// TIA Portal V20 export
FUNCTION_BLOCK "LER_ServoPress"   // FB220, LAD
// stored: Access Published, MemoryReserve 100, SetENOAutomatically false
   VAR_INPUT
      enable : Bool;
      enableManualCmds : Bool;
      interlockHome : Bool;
      interlockRunSequence : Bool;
      interlockJogForward : Bool;
      interlockJogBackward : Bool;
   END_VAR
   VAR_OUTPUT
      error : Bool;
      status : Word;
   END_VAR
   VAR_IN_OUT
      configuration : "LER_typeServoPressConfiguration";
      moduleInterface : "LER_typeServoPressInterface";
      controlNode : "LER_typeServoPressControlNode";
   END_VAR
   VAR
      statProfinetInput { ExternalAccessible := 'False'; ExternalVisible := 'False'; ExternalWritable := 'False'} : "LER_typeServoPress20ByteIn";
      statProfinetOutput { ExternalAccessible := 'False'; ExternalVisible := 'False'; ExternalWritable := 'False'} : "LER_typeServoPress20ByteOut";
      statMonitoring { ExternalAccessible := 'False'; ExternalVisible := 'False'; ExternalWritable := 'False'} : "LER_typeServoPressMonitoring";
      statConfig { ExternalAccessible := 'False'; ExternalVisible := 'False'; ExternalWritable := 'False'} : "LER_typeServoPressConfiguration";
      statRetValInt { ExternalAccessible := 'False'; ExternalVisible := 'False'; ExternalWritable := 'False'} : Array[1..#count] of Int;
      statRetValWord { ExternalAccessible := 'False'; ExternalVisible := 'False'; ExternalWritable := 'False'} : Array[1..#count] of Word;
      statTonTimer { ExternalAccessible := 'False'; ExternalVisible := 'False'; ExternalWritable := 'False'} : Array[0..99] of TON_TIME;
      statConfigCheck { ExternalAccessible := 'False'; ExternalVisible := 'False'; ExternalWritable := 'False'} : Array[0..19] of Bool;
      statConfigHold { ExternalAccessible := 'False'; ExternalVisible := 'False'; ExternalWritable := 'False'} : Array[0..19] of Bool;
      statServoAlarm { ExternalAccessible := 'False'; ExternalVisible := 'False'; ExternalWritable := 'False'} : Struct
         alarmState_0 : Array[0..7] of Bool;
         alarmState_1 : Array[0..7] of Bool;
         alarmState_2 : Array[0..7] of Bool;
         alarmState_3 : Array[0..7] of Bool;
         alarmState_4 : Array[0..7] of Bool;
         alarmState_5 : Array[0..7] of Bool;
         alarmState_6 : Array[0..7] of Bool;
         alarmState_7 : Array[0..7] of Bool;
      END_STRUCT;
      statStep { ExternalAccessible := 'False'; ExternalVisible := 'False'; ExternalWritable := 'False'} : Int;
      statConfigBusy { ExternalAccessible := 'False'; ExternalVisible := 'False'; ExternalWritable := 'False'} : Bool;
      statAckCheck { ExternalAccessible := 'False'; ExternalVisible := 'False'; ExternalWritable := 'False'} : Bool;
      statStop { ExternalAccessible := 'False'; ExternalVisible := 'False'; ExternalWritable := 'False'} : Bool;
   END_VAR
   VAR_TEMP
      tempRetVal : Array[1..#count] of Int;
      tempIndex : Int;
      tempSequenceEnd : Bool;
   END_VAR
   VAR CONSTANT
      False : Bool := False;
      delayTime : Time := T#3s;
      count : Int := 2;
      statusNoErrorOccurred : Word := 16#0000;   // No error occurred.
      errStatusAlarm : Word := 16#8000;
      errStatusSeq : Word := 16#8001;
      errStatusServo : Word := 16#8002;
      errHwdNotConfigured : Word := 16#8090;   // You have not configured a module for the specified hardware identifier or You have ignored the restriction concerning the length of consistent data, or you have not specified a hardware identifier as an address at parameter LADDR
      errRecordDataType : Word := 16#8092;   // Non-supported data type in the RECORD parameter.
      errNoDpProfinetIoModule : Word := 16#8093;   // No DP module/PROFINET IO device from which you can read consistent data exists for the hardware identifier specified in LADDR . This error code also occurs if the module addressed by means of LADDR does not have inputs.
      errIoAccessPermission : Word := 16#80A0;   // An access error was detected when accessing the I/O.
      errRecordLengthInsufficient : Word := 16#80B1;   // The length of the specified destination area at parameter RECORD is shorter than the configured user data length.
      errDataNotReceived : Word := 16#80C0;   // The data have not been read yet.
   END_VAR
   // // statServoAlarm.alarmState_0[0] : ALARM_SETUP_MISMATCH
   // // statServoAlarm.alarmState_0[1] : ALARM_X_SENSOR_CALIBRATION
   // // statServoAlarm.alarmState_0[2] : ALARM_Y_SENSOR_CALIBRATION
   // // statServoAlarm.alarmState_0[3] : ALARM_SENSOR_TEST
   // // statServoAlarm.alarmState_0[4] : ALARM_SENSOR_TEST_WARNING
   // // statServoAlarm.alarmState_0[5] : ALARM_OVER_PIEZO_RANGE
   // // statServoAlarm.alarmState_0[6] : ALARM_NO_EO_CONFIGURED
   // // statServoAlarm.alarmState_0[7] : ALARM_SETUO_MISMATCH_WARNING
   // // statServoAlarm.alarmState_1[0] : reserved
   // // statServoAlarm.alarmState_1[1] : reserved
   // // statServoAlarm.alarmState_1[2] : ALARM_INACTIVE_MP_SELECTED
   // // statServoAlarm.alarmState_1[3] : ALARM_NOK_IN_SEQUENCE
   // // statServoAlarm.alarmState_1[4] : ALARM_NOK_IN_SEQUENCE_WARNING
   // // statServoAlarm.alarmState_1[5] : ALARM_LOST_CYCLES
   // // statServoAlarm.alarmState_1[6] : ALARM_LOST_CYCLES_WARNING
   // // statServoAlarm.alarmState_1[7] : ALARM_NOK_PERCENTAGE_EXCEEDED
   // // statServoAlarm.alarmState_2[0] : ALARM_ENVELOPE_TREND
   // // statServoAlarm.alarmState_2[1] : ALARM_ENVELOPE_WARNING
   // // statServoAlarm.alarmState_2[2] : ALARM_SELFTEST_STRAIN_GAGE_NOK
   // // statServoAlarm.alarmState_2[3] : ALARM_DIG_IO_SHORT_CIRCUIT
   // // statServoAlarm.alarmState_2[4] : ALARM_SELFTEST_5V_SENSOR_POWER
   // // statServoAlarm.alarmState_2[5] : ALARM_SELFTEST_24V_SENSOR_POWER
   // // statServoAlarm.alarmState_2[6] : ALARM_SAMBA_NO_NETWORK_WARNING
   // // statServoAlarm.alarmState_2[7] : ALARM_SAMBA_MEMORY_FULL
   // // statServoAlarm.alarmState_3[0] : ALARM_SAMBA_MEMORY_FULL_WARNING
   // // statServoAlarm.alarmState_3[1] : ALARM_MEMORY_CARD_FULL_WARNING
   // // statServoAlarm.alarmState_3[2] : ALARM_FIFO_FULL
   // // statServoAlarm.alarmState_3[3] : ALARM_FIFO_FULL_WARNING
   // // statServoAlarm.alarmState_3[4] : ALARM_READING_UV_WITHOUT_DESCRIPTION
   // // statServoAlarm.alarmState_3[5] : ALARM_POWER_COULD_NOT_BE_ENABLED
   // // statServoAlarm.alarmState_3[6] : ALARM_MULTIPLE_PLC_MOVEMENT_COMMANDS
   // // statServoAlarm.alarmState_3[7] : ALARM_SEQ_CALCULATOR_IN_MEASUREMENT
   // // statServoAlarm.alarmState_4[0] : ALARM_SEQ_DYNAMIC_CALC_DIV_BY_ZERO
   // // statServoAlarm.alarmState_4[1] : ALARM_SEQ_DYNAMIC_FORCE_TRIGGER_NOT_
   // // statServoAlarm.alarmState_4[2] : ALARM_SEQ_POSITION_SET_OUTSIDE_THE_RA
   // // statServoAlarm.alarmState_4[3] : ALARM_SERVO_CONTROLLER_CONNECTION
   // // statServoAlarm.alarmState_4[4] : ALARM_SERVO_CONTROLLER_ERROR
   // // statServoAlarm.alarmState_4[5] : ALARM_SERVO_CONTROLLER_WARNING
   // // statServoAlarm.alarmState_4[6] : ALARM_SERVO_MAX_FORCE_TRIGGER
   // // statServoAlarm.alarmState_4[7] : ALARM_SERVO_DISPL_OVERRANGE
   // // statServoAlarm.alarmState_5[0] : ALARM_SERVO_STOP_EXT_SIGNAL_NOT_REACHED
   // // statServoAlarm.alarmState_5[1] : ALARM_SEQ_DYNAMIC_ZERO_MOTION_SPEED
   // // statServoAlarm.alarmState_5[2] : ALARM_ADC_2_DAC_ADC_FACTOR_IS_OUT_OF_RANGE
   // // statServoAlarm.alarmState_5[3] : ALARM_SEQ_SPEED_SET_OUTSIDE_THE_RANG
   // // statServoAlarm.alarmState_5[4] : ALARM_JOG_SPEED_IS_OUT_OF_RANGE
   // // statServoAlarm.alarmState_5[5] : ALARM_BRAKETEST_FAILED
   // // statServoAlarm.alarmState_5[6] : ALARM_SEQ_DYNAMIC_UNKNOWN_ERROR
   // // statServoAlarm.alarmState_5[7] : ALARM_SEQ_DIGITAL_INPUT_TIMOUT_BEFORE_SIGNAL
   VAR_TEMP   // added for the SCL form of the ladder/FBD networks
      _w1 : Bool;
      _w2 : Bool;
      _w3 : Bool;
   END_VAR
BEGIN

REGION Network 1: DP Read
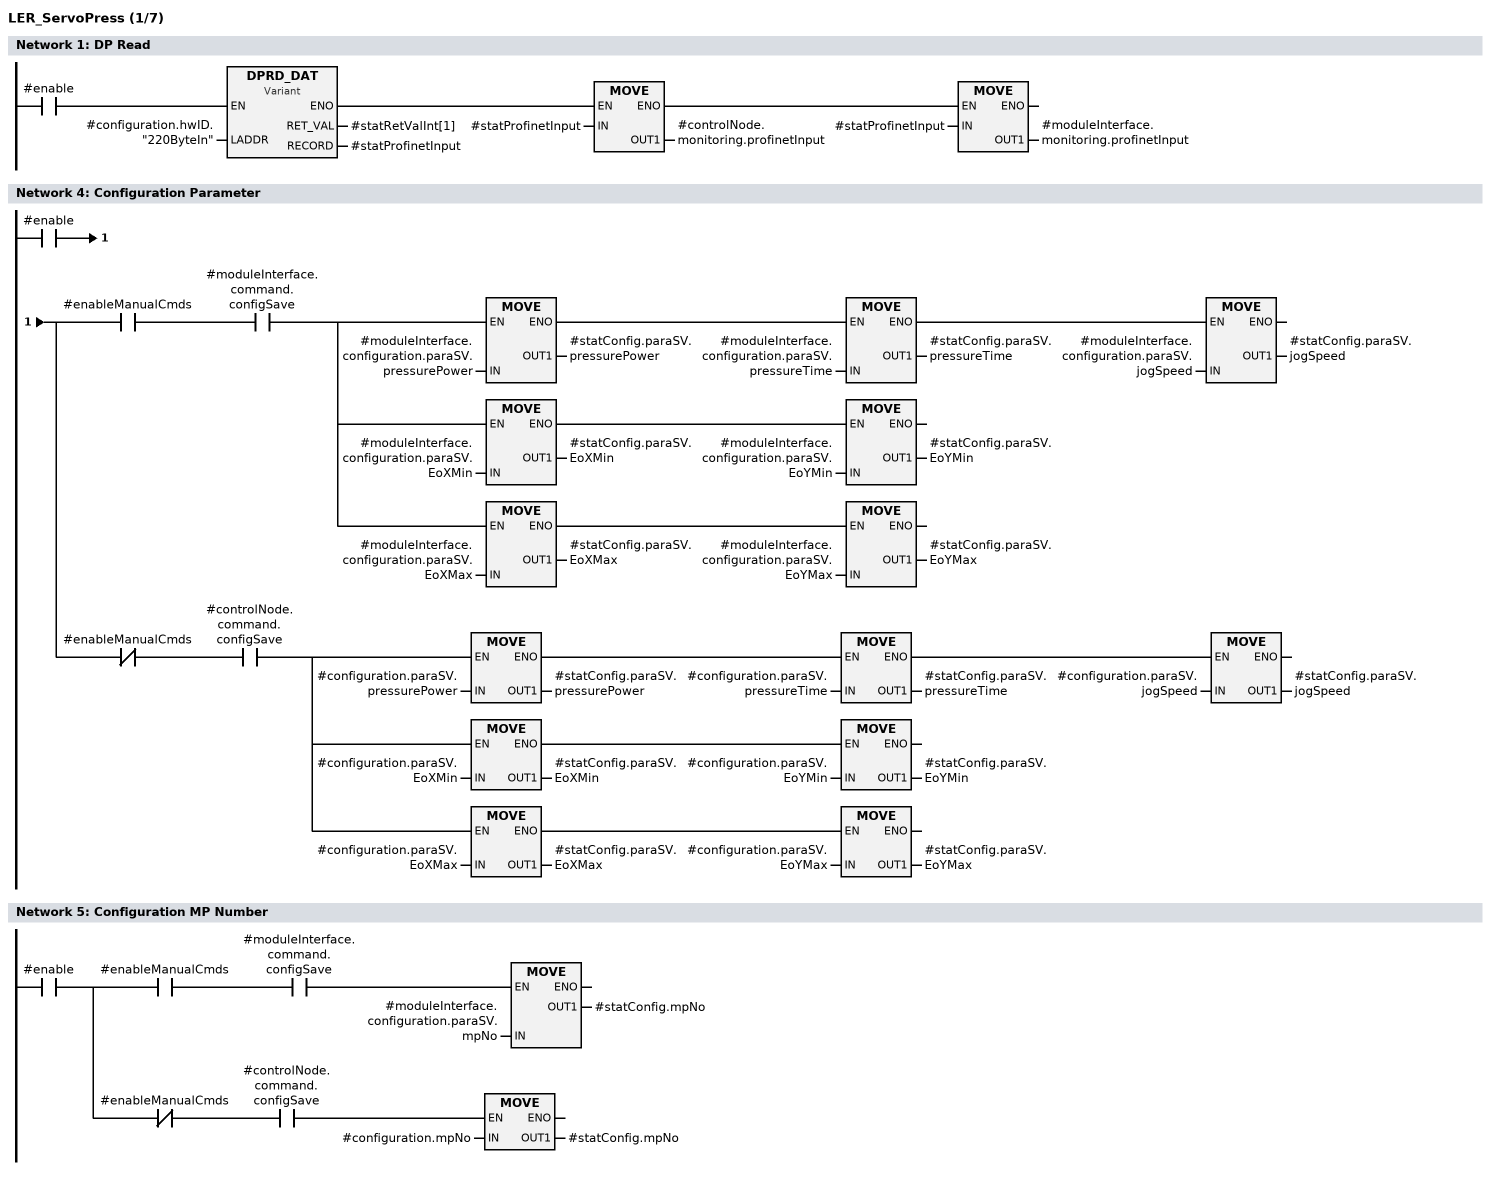
   RUNG wire#powerrail
      Contact( #enable )
      { S7_Templates := "[ptr_type := Variant, laddr_type := HW_IO]" } DPRD_DAT(LADDR := #configuration.hwID."220ByteIn", RET_VAL => #statRetValInt[1], RECORD => #statProfinetInput)
      Move(in := #statProfinetInput, out1 => #controlNode.monitoring.profinetInput)
      Move(in := #statProfinetInput, out1 => #moduleInterface.monitoring.profinetInput)
   END_RUNG
   // the same network as SCL:
   #statRetValInt[1] := DPRD_DAT(EN := #enable,
                           LADDR := #configuration.hwID."220ByteIn",
                           RECORD => #statProfinetInput,
                           ENO => #_w1);
   IF #_w1 THEN
       #controlNode.monitoring.profinetInput := #statProfinetInput;
       #moduleInterface.monitoring.profinetInput := #statProfinetInput;
   END_IF;
END_REGION

REGION Network 2 (SCL): Input Mapping
   REGION Input mapping

   #statMonitoring.profinetInput := #statProfinetInput;

   END_REGION
END_REGION

REGION Network 3 (SCL): Error Status
   REGION Error check

       IF #enable THEN
           IF #statRetValInt <> #tempRetVal THEN
               FOR #tempIndex := 1 TO #count DO
                   #statRetValWord[#tempIndex] := INT_TO_WORD(#statRetValInt[#tempIndex]); // convert the return value of DPRD, DPWR form int to word
                   CASE #statRetValWord[#tempIndex] OF

                       #errHwdNotConfigured:
                           #status := #errHwdNotConfigured;

                       #errRecordDataType:
                           #status := #errRecordDataType;

                       #errNoDpProfinetIoModule:
                           #status := #errNoDpProfinetIoModule;

                       #errIoAccessPermission:
                           #status := #errIoAccessPermission;

                       #errRecordLengthInsufficient:
                           #status := #errRecordLengthInsufficient;

                       #errDataNotReceived:
                           #status := #errDataNotReceived;
                   END_CASE;
               END_FOR;

           ELSIF #statMonitoring.profinetInput.ALARM THEN
               #status := #errStatusAlarm;

           ELSIF #statMonitoring.profinetInput."SEQUENCE-ERROR" THEN
               #status := #errStatusSeq;

           ELSIF #statMonitoring.profinetInput."SERVO-ERROR" THEN
               #status := #errStatusServo;

           ELSE
               #status := #statusNoErrorOccurred;
           END_IF;
       ELSE
           #status := #statusNoErrorOccurred;
       END_IF;

       #error := #status <> 0;

   END_REGION
END_REGION

REGION Network 4: Configuration Parameter
   RUNG wire#powerrail
      Contact( #enable )
      wire#w1
      Contact( #enableManualCmds )
      Contact( #moduleInterface.command.configSave )
      wire#w2
      Move(in := #moduleInterface.configuration.paraSV.pressurePower, out1 => #statConfig.paraSV.pressurePower)
      Move(in := #moduleInterface.configuration.paraSV.pressureTime, out1 => #statConfig.paraSV.pressureTime)
      Move(in := #moduleInterface.configuration.paraSV.jogSpeed, out1 => #statConfig.paraSV.jogSpeed)
   END_RUNG
   RUNG wire#w2
      Move(in := #moduleInterface.configuration.paraSV.EoXMin, out1 => #statConfig.paraSV.EoXMin)
      Move(in := #moduleInterface.configuration.paraSV.EoYMin, out1 => #statConfig.paraSV.EoYMin)
   END_RUNG
   RUNG wire#w2
      Move(in := #moduleInterface.configuration.paraSV.EoXMax, out1 => #statConfig.paraSV.EoXMax)
      Move(in := #moduleInterface.configuration.paraSV.EoYMax, out1 => #statConfig.paraSV.EoYMax)
   END_RUNG
   RUNG wire#w1
      I_Contact( #enableManualCmds )
      Contact( #controlNode.command.configSave )
      wire#w3
      Move(in := #configuration.paraSV.pressurePower, out1 => #statConfig.paraSV.pressurePower)
      Move(in := #configuration.paraSV.pressureTime, out1 => #statConfig.paraSV.pressureTime)
      Move(in := #configuration.paraSV.jogSpeed, out1 => #statConfig.paraSV.jogSpeed)
   END_RUNG
   RUNG wire#w3
      Move(in := #configuration.paraSV.EoXMin, out1 => #statConfig.paraSV.EoXMin)
      Move(in := #configuration.paraSV.EoYMin, out1 => #statConfig.paraSV.EoYMin)
   END_RUNG
   RUNG wire#w3
      Move(in := #configuration.paraSV.EoXMax, out1 => #statConfig.paraSV.EoXMax)
      Move(in := #configuration.paraSV.EoYMax, out1 => #statConfig.paraSV.EoYMax)
   END_RUNG
   // the same network as SCL:
   IF #enable AND #enableManualCmds AND #moduleInterface.command.configSave THEN
       #statConfig.paraSV.pressurePower := #moduleInterface.configuration.paraSV.pressurePower;
       #statConfig.paraSV.pressureTime := #moduleInterface.configuration.paraSV.pressureTime;
       #statConfig.paraSV.jogSpeed := #moduleInterface.configuration.paraSV.jogSpeed;
       #statConfig.paraSV.EoXMin := #moduleInterface.configuration.paraSV.EoXMin;
       #statConfig.paraSV.EoYMin := #moduleInterface.configuration.paraSV.EoYMin;
       #statConfig.paraSV.EoXMax := #moduleInterface.configuration.paraSV.EoXMax;
       #statConfig.paraSV.EoYMax := #moduleInterface.configuration.paraSV.EoYMax;
   END_IF;
   IF #enable AND NOT #enableManualCmds AND #controlNode.command.configSave THEN
       #statConfig.paraSV.pressurePower := #configuration.paraSV.pressurePower;
       #statConfig.paraSV.pressureTime := #configuration.paraSV.pressureTime;
       #statConfig.paraSV.jogSpeed := #configuration.paraSV.jogSpeed;
       #statConfig.paraSV.EoXMin := #configuration.paraSV.EoXMin;
       #statConfig.paraSV.EoYMin := #configuration.paraSV.EoYMin;
       #statConfig.paraSV.EoXMax := #configuration.paraSV.EoXMax;
       #statConfig.paraSV.EoYMax := #configuration.paraSV.EoYMax;
   END_IF;
END_REGION

REGION Network 5: Configuration MP Number
   RUNG wire#powerrail
      Contact( #enable )
      wire#w1
      Contact( #enableManualCmds )
      Contact( #moduleInterface.command.configSave )
      Move(in := #moduleInterface.configuration.paraSV.mpNo, out1 => #statConfig.mpNo)
   END_RUNG
   RUNG wire#w1
      I_Contact( #enableManualCmds )
      Contact( #controlNode.command.configSave )
      Move(in := #configuration.mpNo, out1 => #statConfig.mpNo)
   END_RUNG
   // the same network as SCL:
   IF #enable AND #enableManualCmds AND #moduleInterface.command.configSave THEN
       #statConfig.mpNo := #moduleInterface.configuration.paraSV.mpNo;
   END_IF;
   IF #enable AND NOT #enableManualCmds AND #controlNode.command.configSave THEN
       #statConfig.mpNo := #configuration.mpNo;
   END_IF;
END_REGION

REGION Network 6: Configuration Sequence Number
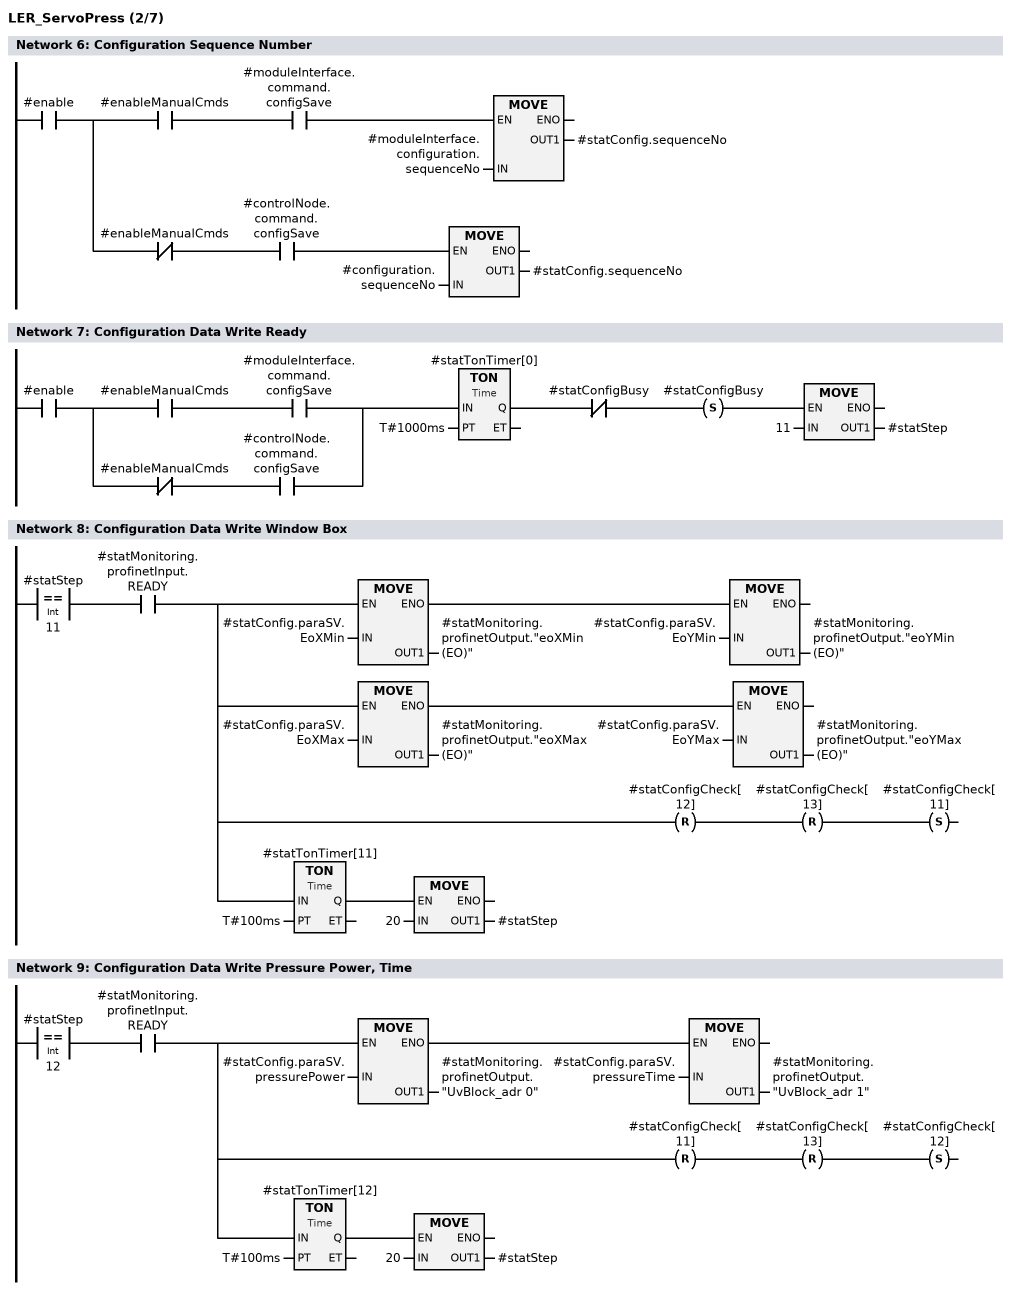
   RUNG wire#powerrail
      Contact( #enable )
      wire#w1
      Contact( #enableManualCmds )
      Contact( #moduleInterface.command.configSave )
      Move(in := #moduleInterface.configuration.sequenceNo, out1 => #statConfig.sequenceNo)
   END_RUNG
   RUNG wire#w1
      I_Contact( #enableManualCmds )
      Contact( #controlNode.command.configSave )
      Move(in := #configuration.sequenceNo, out1 => #statConfig.sequenceNo)
   END_RUNG
   // the same network as SCL:
   IF #enable AND #enableManualCmds AND #moduleInterface.command.configSave THEN
       #statConfig.sequenceNo := #moduleInterface.configuration.sequenceNo;
   END_IF;
   IF #enable AND NOT #enableManualCmds AND #controlNode.command.configSave THEN
       #statConfig.sequenceNo := #configuration.sequenceNo;
   END_IF;
END_REGION

REGION Network 7: Configuration Data Write Ready
   RUNG wire#powerrail
      Contact( #enable )
      wire#w1
      Contact( #enableManualCmds )
      Contact( #moduleInterface.command.configSave )
      wire#w2
      { S7_Templates := "time_type := Time" } #statTonTimer[0].TON(pt := T#1000ms, et =>)
      I_Contact( #statConfigBusy )
      S_Coil( #statConfigBusy )
      Move(in := 11, out1 => #statStep)
   END_RUNG
   RUNG wire#w1
      I_Contact( #enableManualCmds )
      Contact( #controlNode.command.configSave )
   END_RUNG wire#w2
   // the same network as SCL:
   #statTonTimer[0].TON(IN := #enable AND ((#enableManualCmds AND #moduleInterface.command.configSave) OR (NOT #enableManualCmds AND #controlNode.command.configSave)),
                        PT := T#1000ms);
   #_w1 := #statTonTimer[0].Q AND NOT #statConfigBusy;
   IF #_w1 THEN
       #statConfigBusy := TRUE;
       #statStep := 11;
   END_IF;
END_REGION

REGION Network 8: Configuration Data Write Window Box
   RUNG wire#powerrail
      { S7_Templates := "SrcType := Int" } EQ_Contact(in1 := #statStep, in2 := 11)
      Contact( #statMonitoring.profinetInput.READY )
      wire#w1
      Move(in := #statConfig.paraSV.EoXMin, out1 => #statMonitoring.profinetOutput."eoXMin (EO)")
      Move(in := #statConfig.paraSV.EoYMin, out1 => #statMonitoring.profinetOutput."eoYMin (EO)")
   END_RUNG
   RUNG wire#w1
      Move(in := #statConfig.paraSV.EoXMax, out1 => #statMonitoring.profinetOutput."eoXMax (EO)")
      Move(in := #statConfig.paraSV.EoYMax, out1 => #statMonitoring.profinetOutput."eoYMax (EO)")
   END_RUNG
   RUNG wire#w1
      R_Coil( #statConfigCheck[12] )
      R_Coil( #statConfigCheck[13] )
      S_Coil( #statConfigCheck[11] )
   END_RUNG
   RUNG wire#w1
      { S7_Templates := "time_type := Time" } #statTonTimer[11].TON(pt := T#100ms, et =>)
      Move(in := 20, out1 => #statStep)
   END_RUNG
   // the same network as SCL:
   #_w1 := (#statStep = 11) AND #statMonitoring.profinetInput.READY;
   IF #_w1 THEN
       #statMonitoring.profinetOutput."eoXMin (EO)" := #statConfig.paraSV.EoXMin;
       #statMonitoring.profinetOutput."eoYMin (EO)" := #statConfig.paraSV.EoYMin;
       #statMonitoring.profinetOutput."eoXMax (EO)" := #statConfig.paraSV.EoXMax;
       #statMonitoring.profinetOutput."eoYMax (EO)" := #statConfig.paraSV.EoYMax;
       #statConfigCheck[12] := FALSE;
       #statConfigCheck[13] := FALSE;
       #statConfigCheck[11] := TRUE;
   END_IF;
   #statTonTimer[11].TON(IN := #_w1, PT := T#100ms);
   IF #statTonTimer[11].Q THEN #statStep := 20; END_IF;
END_REGION

REGION Network 9: Configuration Data Write Pressure Power, Time
   RUNG wire#powerrail
      { S7_Templates := "SrcType := Int" } EQ_Contact(in1 := #statStep, in2 := 12)
      Contact( #statMonitoring.profinetInput.READY )
      wire#w1
      Move(in := #statConfig.paraSV.pressurePower, out1 => #statMonitoring.profinetOutput."UvBlock_adr 0")
      Move(in := #statConfig.paraSV.pressureTime, out1 => #statMonitoring.profinetOutput."UvBlock_adr 1")
   END_RUNG
   RUNG wire#w1
      R_Coil( #statConfigCheck[11] )
      R_Coil( #statConfigCheck[13] )
      S_Coil( #statConfigCheck[12] )
   END_RUNG
   RUNG wire#w1
      { S7_Templates := "time_type := Time" } #statTonTimer[12].TON(pt := T#100ms, et =>)
      Move(in := 20, out1 => #statStep)
   END_RUNG
   // the same network as SCL:
   #_w1 := (#statStep = 12) AND #statMonitoring.profinetInput.READY;
   IF #_w1 THEN
       #statMonitoring.profinetOutput."UvBlock_adr 0" := #statConfig.paraSV.pressurePower;
       #statMonitoring.profinetOutput."UvBlock_adr 1" := #statConfig.paraSV.pressureTime;
       #statConfigCheck[11] := FALSE;
       #statConfigCheck[13] := FALSE;
       #statConfigCheck[12] := TRUE;
   END_IF;
   #statTonTimer[12].TON(IN := #_w1, PT := T#100ms);
   IF #statTonTimer[12].Q THEN #statStep := 20; END_IF;
END_REGION

REGION Network 10: Configuration Data Write Jog Speed
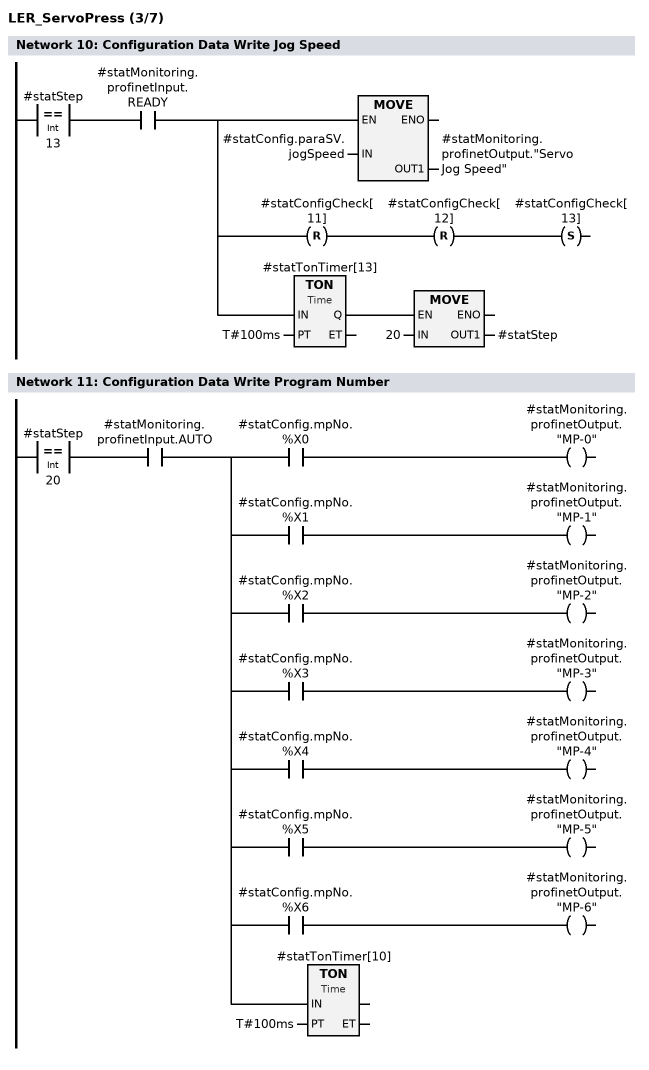
   RUNG wire#powerrail
      { S7_Templates := "SrcType := Int" } EQ_Contact(in1 := #statStep, in2 := 13)
      Contact( #statMonitoring.profinetInput.READY )
      wire#w1
      Move(in := #statConfig.paraSV.jogSpeed, out1 => #statMonitoring.profinetOutput."Servo Jog Speed")
   END_RUNG
   RUNG wire#w1
      R_Coil( #statConfigCheck[11] )
      R_Coil( #statConfigCheck[12] )
      S_Coil( #statConfigCheck[13] )
   END_RUNG
   RUNG wire#w1
      { S7_Templates := "time_type := Time" } #statTonTimer[13].TON(pt := T#100ms, et =>)
      Move(in := 20, out1 => #statStep)
   END_RUNG
   // the same network as SCL:
   #_w1 := (#statStep = 13) AND #statMonitoring.profinetInput.READY;
   IF #_w1 THEN
       #statMonitoring.profinetOutput."Servo Jog Speed" := #statConfig.paraSV.jogSpeed;
       #statConfigCheck[11] := FALSE;
       #statConfigCheck[12] := FALSE;
       #statConfigCheck[13] := TRUE;
   END_IF;
   #statTonTimer[13].TON(IN := #_w1, PT := T#100ms);
   IF #statTonTimer[13].Q THEN #statStep := 20; END_IF;
END_REGION

REGION Network 11: Configuration Data Write Program Number
   RUNG wire#powerrail
      { S7_Templates := "SrcType := Int" } EQ_Contact(in1 := #statStep, in2 := 20)
      Contact( #statMonitoring.profinetInput.AUTO )
      wire#w1
      Contact( #statConfig.mpNo.%X0 )
      Coil( #statMonitoring.profinetOutput."MP-0" )
   END_RUNG
   RUNG wire#w1
      Contact( #statConfig.mpNo.%X1 )
      Coil( #statMonitoring.profinetOutput."MP-1" )
   END_RUNG
   RUNG wire#w1
      Contact( #statConfig.mpNo.%X2 )
      Coil( #statMonitoring.profinetOutput."MP-2" )
   END_RUNG
   RUNG wire#w1
      Contact( #statConfig.mpNo.%X3 )
      Coil( #statMonitoring.profinetOutput."MP-3" )
   END_RUNG
   RUNG wire#w1
      Contact( #statConfig.mpNo.%X4 )
      Coil( #statMonitoring.profinetOutput."MP-4" )
   END_RUNG
   RUNG wire#w1
      Contact( #statConfig.mpNo.%X5 )
      Coil( #statMonitoring.profinetOutput."MP-5" )
   END_RUNG
   RUNG wire#w1
      Contact( #statConfig.mpNo.%X6 )
      Coil( #statMonitoring.profinetOutput."MP-6" )
   END_RUNG
   RUNG wire#w1
      { S7_Templates := "time_type := Time" } #statTonTimer[10].TON(pt := T#100ms, et =>)
   END_RUNG
   // the same network as SCL:
   #_w1 := (#statStep = 20) AND #statMonitoring.profinetInput.AUTO;
   #statMonitoring.profinetOutput."MP-0" := #_w1 AND #statConfig.mpNo.%X0;
   #statMonitoring.profinetOutput."MP-1" := #_w1 AND #statConfig.mpNo.%X1;
   #statMonitoring.profinetOutput."MP-2" := #_w1 AND #statConfig.mpNo.%X2;
   #statMonitoring.profinetOutput."MP-3" := #_w1 AND #statConfig.mpNo.%X3;
   #statMonitoring.profinetOutput."MP-4" := #_w1 AND #statConfig.mpNo.%X4;
   #statMonitoring.profinetOutput."MP-5" := #_w1 AND #statConfig.mpNo.%X5;
   #statMonitoring.profinetOutput."MP-6" := #_w1 AND #statConfig.mpNo.%X6;
   #statTonTimer[10].TON(IN := #_w1, PT := T#100ms);
END_REGION

REGION Network 12: Configuration Data Write CFG
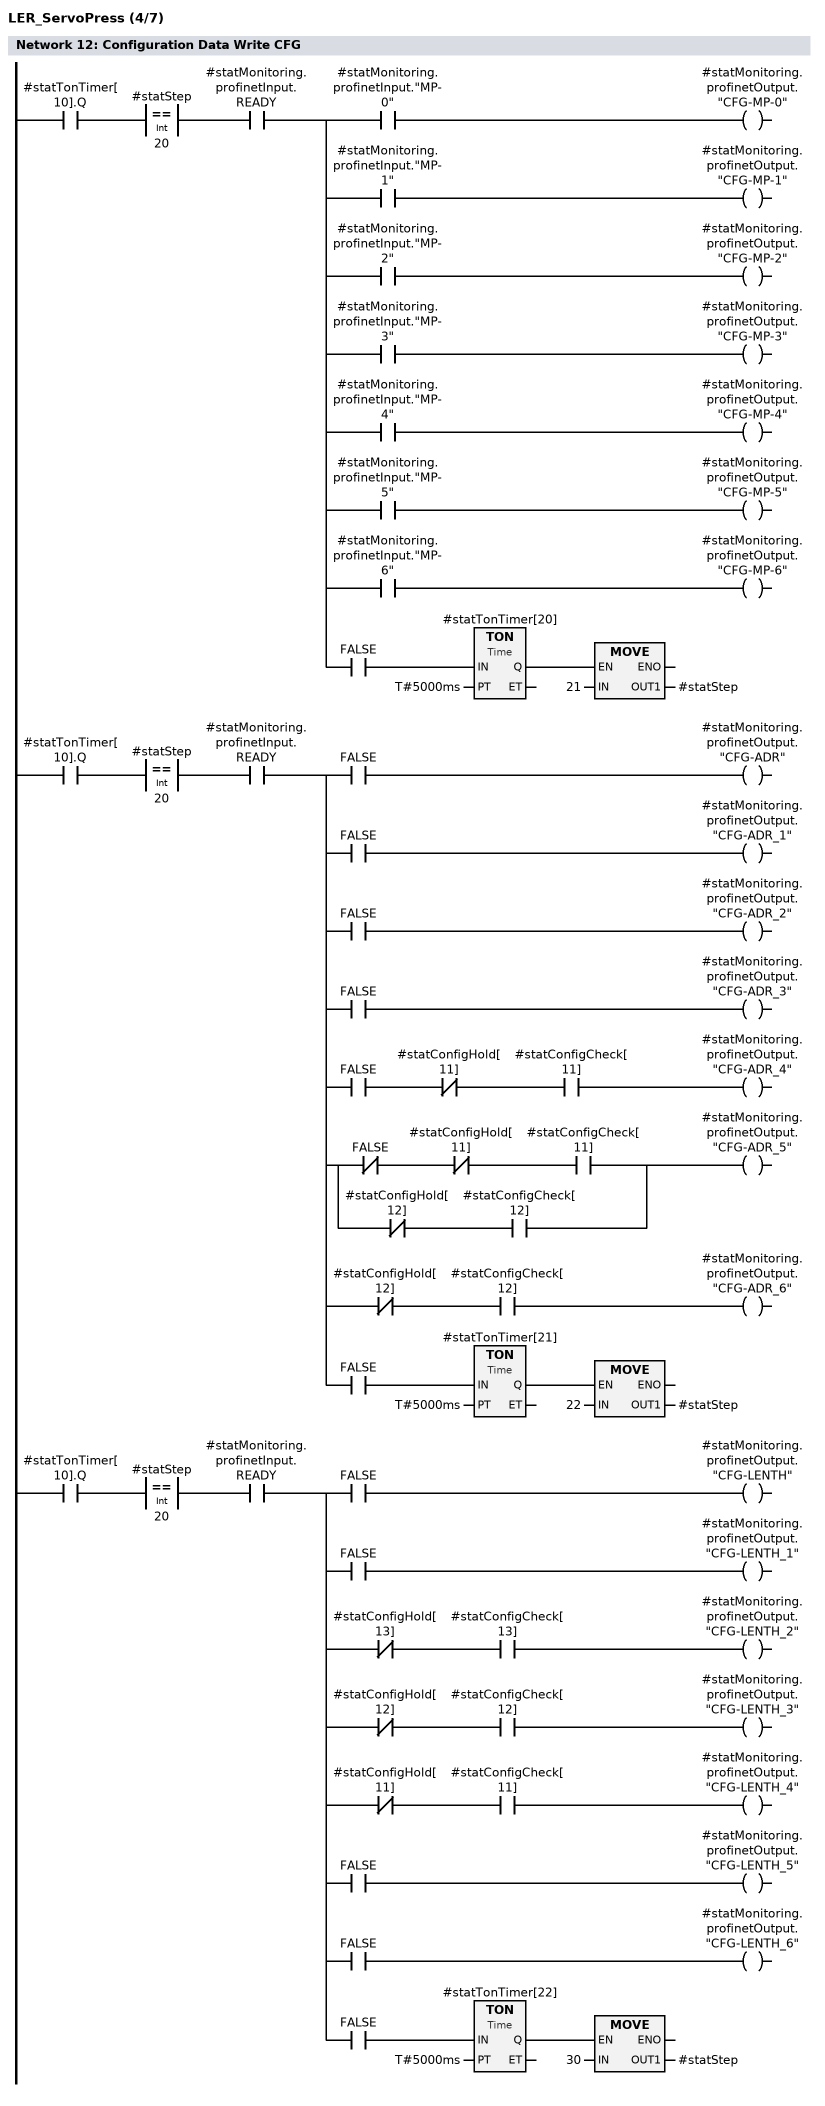
   RUNG wire#powerrail
      Contact( #statTonTimer[10].Q )
      { S7_Templates := "SrcType := Int" } EQ_Contact(in1 := #statStep, in2 := 20)
      Contact( #statMonitoring.profinetInput.READY )
      wire#w1
      Contact( #statMonitoring.profinetInput."MP-0" )
      Coil( #statMonitoring.profinetOutput."CFG-MP-0" )
   END_RUNG
   RUNG wire#w1
      Contact( #statMonitoring.profinetInput."MP-1" )
      Coil( #statMonitoring.profinetOutput."CFG-MP-1" )
   END_RUNG
   RUNG wire#w1
      Contact( #statMonitoring.profinetInput."MP-2" )
      Coil( #statMonitoring.profinetOutput."CFG-MP-2" )
   END_RUNG
   RUNG wire#w1
      Contact( #statMonitoring.profinetInput."MP-3" )
      Coil( #statMonitoring.profinetOutput."CFG-MP-3" )
   END_RUNG
   RUNG wire#w1
      Contact( #statMonitoring.profinetInput."MP-4" )
      Coil( #statMonitoring.profinetOutput."CFG-MP-4" )
   END_RUNG
   RUNG wire#w1
      Contact( #statMonitoring.profinetInput."MP-5" )
      Coil( #statMonitoring.profinetOutput."CFG-MP-5" )
   END_RUNG
   RUNG wire#w1
      Contact( #statMonitoring.profinetInput."MP-6" )
      Coil( #statMonitoring.profinetOutput."CFG-MP-6" )
   END_RUNG
   RUNG wire#w1
      Contact( FALSE )
      { S7_Templates := "time_type := Time" } #statTonTimer[20].TON(pt := T#5000ms, et =>)
      Move(in := 21, out1 => #statStep)
   END_RUNG
   RUNG wire#powerrail
      Contact( #statTonTimer[10].Q )
      { S7_Templates := "SrcType := Int" } EQ_Contact(in1 := #statStep, in2 := 20)
      Contact( #statMonitoring.profinetInput.READY )
      wire#w2
      Contact( FALSE )
      Coil( #statMonitoring.profinetOutput."CFG-ADR" )
   END_RUNG
   RUNG wire#w2
      Contact( FALSE )
      Coil( #statMonitoring.profinetOutput."CFG-ADR_1" )
   END_RUNG
   RUNG wire#w2
      Contact( FALSE )
      Coil( #statMonitoring.profinetOutput."CFG-ADR_2" )
   END_RUNG
   RUNG wire#w2
      Contact( FALSE )
      Coil( #statMonitoring.profinetOutput."CFG-ADR_3" )
   END_RUNG
   RUNG wire#w2
      Contact( FALSE )
      I_Contact( #statConfigHold[11] )
      Contact( #statConfigCheck[11] )
      Coil( #statMonitoring.profinetOutput."CFG-ADR_4" )
   END_RUNG
   RUNG wire#w2
      I_Contact( FALSE )
      I_Contact( #statConfigHold[11] )
      Contact( #statConfigCheck[11] )
      wire#w3
      Coil( #statMonitoring.profinetOutput."CFG-ADR_5" )
   END_RUNG
   RUNG wire#w2
      I_Contact( #statConfigHold[12] )
      Contact( #statConfigCheck[12] )
   END_RUNG wire#w3
   RUNG wire#w2
      I_Contact( #statConfigHold[12] )
      Contact( #statConfigCheck[12] )
      Coil( #statMonitoring.profinetOutput."CFG-ADR_6" )
   END_RUNG
   RUNG wire#w2
      Contact( FALSE )
      { S7_Templates := "time_type := Time" } #statTonTimer[21].TON(pt := T#5000ms, et =>)
      Move(in := 22, out1 => #statStep)
   END_RUNG
   RUNG wire#powerrail
      Contact( #statTonTimer[10].Q )
      { S7_Templates := "SrcType := Int" } EQ_Contact(in1 := #statStep, in2 := 20)
      Contact( #statMonitoring.profinetInput.READY )
      wire#w4
      Contact( FALSE )
      Coil( #statMonitoring.profinetOutput."CFG-LENTH" )
   END_RUNG
   RUNG wire#w4
      Contact( FALSE )
      Coil( #statMonitoring.profinetOutput."CFG-LENTH_1" )
   END_RUNG
   RUNG wire#w4
      I_Contact( #statConfigHold[13] )
      Contact( #statConfigCheck[13] )
      Coil( #statMonitoring.profinetOutput."CFG-LENTH_2" )
   END_RUNG
   RUNG wire#w4
      I_Contact( #statConfigHold[12] )
      Contact( #statConfigCheck[12] )
      Coil( #statMonitoring.profinetOutput."CFG-LENTH_3" )
   END_RUNG
   RUNG wire#w4
      I_Contact( #statConfigHold[11] )
      Contact( #statConfigCheck[11] )
      Coil( #statMonitoring.profinetOutput."CFG-LENTH_4" )
   END_RUNG
   RUNG wire#w4
      Contact( FALSE )
      Coil( #statMonitoring.profinetOutput."CFG-LENTH_5" )
   END_RUNG
   RUNG wire#w4
      Contact( FALSE )
      Coil( #statMonitoring.profinetOutput."CFG-LENTH_6" )
   END_RUNG
   RUNG wire#w4
      Contact( FALSE )
      { S7_Templates := "time_type := Time" } #statTonTimer[22].TON(pt := T#5000ms, et =>)
      Move(in := 30, out1 => #statStep)
   END_RUNG
   // the same network as SCL:
   #_w1 := #statTonTimer[10].Q AND (#statStep = 20) AND #statMonitoring.profinetInput.READY;
   #statMonitoring.profinetOutput."CFG-MP-0" := #_w1 AND #statMonitoring.profinetInput."MP-0";
   #statMonitoring.profinetOutput."CFG-MP-1" := #_w1 AND #statMonitoring.profinetInput."MP-1";
   #statMonitoring.profinetOutput."CFG-MP-2" := #_w1 AND #statMonitoring.profinetInput."MP-2";
   #statMonitoring.profinetOutput."CFG-MP-3" := #_w1 AND #statMonitoring.profinetInput."MP-3";
   #statMonitoring.profinetOutput."CFG-MP-4" := #_w1 AND #statMonitoring.profinetInput."MP-4";
   #statMonitoring.profinetOutput."CFG-MP-5" := #_w1 AND #statMonitoring.profinetInput."MP-5";
   #statMonitoring.profinetOutput."CFG-MP-6" := #_w1 AND #statMonitoring.profinetInput."MP-6";
   #statTonTimer[20].TON(IN := #_w1 AND FALSE, PT := T#5000ms);
   IF #statTonTimer[20].Q THEN #statStep := 21; END_IF;
   #_w2 := #statTonTimer[10].Q AND (#statStep = 20) AND #statMonitoring.profinetInput.READY;
   #statMonitoring.profinetOutput."CFG-ADR" := #_w2 AND FALSE;
   #statMonitoring.profinetOutput."CFG-ADR_1" := #_w2 AND FALSE;
   #statMonitoring.profinetOutput."CFG-ADR_2" := #_w2 AND FALSE;
   #statMonitoring.profinetOutput."CFG-ADR_3" := #_w2 AND FALSE;
   #statMonitoring.profinetOutput."CFG-ADR_4" := #_w2 AND FALSE AND NOT #statConfigHold[11] AND #statConfigCheck[11];
   #statMonitoring.profinetOutput."CFG-ADR_5" := #_w2 AND ((NOT FALSE AND NOT #statConfigHold[11] AND #statConfigCheck[11]) OR (NOT #statConfigHold[12] AND #statConfigCheck[12]));
   #statMonitoring.profinetOutput."CFG-ADR_6" := #_w2 AND NOT #statConfigHold[12] AND #statConfigCheck[12];
   #statTonTimer[21].TON(IN := #_w2 AND FALSE, PT := T#5000ms);
   IF #statTonTimer[21].Q THEN #statStep := 22; END_IF;
   #_w3 := #statTonTimer[10].Q AND (#statStep = 20) AND #statMonitoring.profinetInput.READY;
   #statMonitoring.profinetOutput."CFG-LENTH" := #_w3 AND FALSE;
   #statMonitoring.profinetOutput."CFG-LENTH_1" := #_w3 AND FALSE;
   #statMonitoring.profinetOutput."CFG-LENTH_2" := #_w3 AND NOT #statConfigHold[13] AND #statConfigCheck[13];
   #statMonitoring.profinetOutput."CFG-LENTH_3" := #_w3 AND NOT #statConfigHold[12] AND #statConfigCheck[12];
   #statMonitoring.profinetOutput."CFG-LENTH_4" := #_w3 AND NOT #statConfigHold[11] AND #statConfigCheck[11];
   #statMonitoring.profinetOutput."CFG-LENTH_5" := #_w3 AND FALSE;
   #statMonitoring.profinetOutput."CFG-LENTH_6" := #_w3 AND FALSE;
   #statTonTimer[22].TON(IN := #_w3 AND FALSE, PT := T#5000ms);
   IF #statTonTimer[22].Q THEN #statStep := 30; END_IF;
END_REGION

REGION Network 13: Configuration Data Write Start
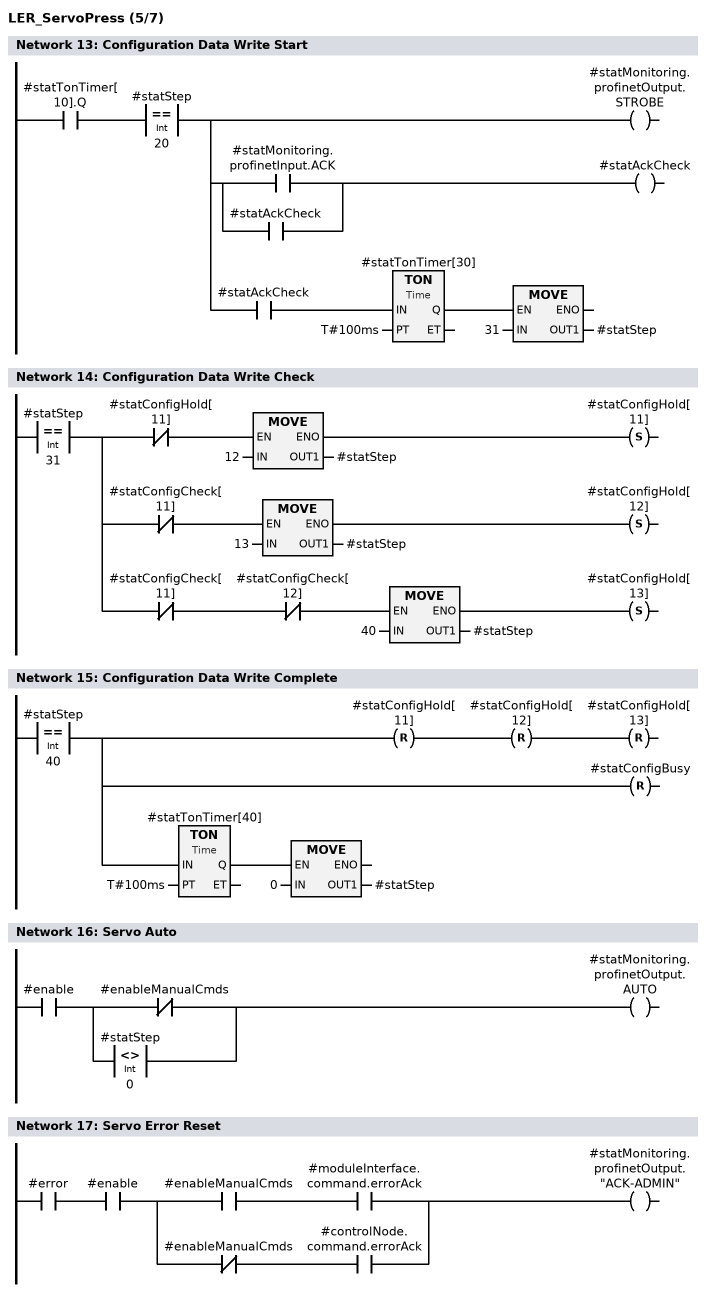
   RUNG wire#powerrail
      Contact( #statTonTimer[10].Q )
      { S7_Templates := "SrcType := Int" } EQ_Contact(in1 := #statStep, in2 := 20)
      wire#w1
      Coil( #statMonitoring.profinetOutput.STROBE )
   END_RUNG
   RUNG wire#w1
      Contact( #statMonitoring.profinetInput.ACK )
      wire#w2
      Coil( #statAckCheck )
   END_RUNG
   RUNG wire#w1
      Contact( #statAckCheck )
   END_RUNG wire#w2
   RUNG wire#w1
      Contact( #statAckCheck )
      { S7_Templates := "time_type := Time" } #statTonTimer[30].TON(pt := T#100ms, et =>)
      Move(in := 31, out1 => #statStep)
   END_RUNG
   // the same network as SCL:
   #statMonitoring.profinetOutput.STROBE := #statTonTimer[10].Q AND (#statStep = 20);
   #statAckCheck := #statMonitoring.profinetOutput.STROBE AND (#statMonitoring.profinetInput.ACK OR #statAckCheck);
   #statTonTimer[30].TON(IN := #statMonitoring.profinetOutput.STROBE AND #statAckCheck, PT := T#100ms);
   IF #statTonTimer[30].Q THEN #statStep := 31; END_IF;
END_REGION

REGION Network 14: Configuration Data Write Check
   RUNG wire#powerrail
      { S7_Templates := "SrcType := Int" } EQ_Contact(in1 := #statStep, in2 := 31)
      wire#w1
      I_Contact( #statConfigHold[11] )
      Move(in := 12, out1 => #statStep)
      S_Coil( #statConfigHold[11] )
   END_RUNG
   RUNG wire#w1
      I_Contact( #statConfigCheck[11] )
      Move(in := 13, out1 => #statStep)
      S_Coil( #statConfigHold[12] )
   END_RUNG
   RUNG wire#w1
      I_Contact( #statConfigCheck[11] )
      I_Contact( #statConfigCheck[12] )
      Move(in := 40, out1 => #statStep)
      S_Coil( #statConfigHold[13] )
   END_RUNG
   // the same network as SCL:
   #_w1 := #statStep = 31;
   IF #_w1 AND NOT #statConfigHold[11] THEN
       #statStep := 12;
       #statConfigHold[11] := TRUE;
   END_IF;
   IF #_w1 AND NOT #statConfigCheck[11] THEN
       #statStep := 13;
       #statConfigHold[12] := TRUE;
   END_IF;
   IF #_w1 AND NOT #statConfigCheck[11] AND NOT #statConfigCheck[12] THEN
       #statStep := 40;
       #statConfigHold[13] := TRUE;
   END_IF;
END_REGION

REGION Network 15: Configuration Data Write Complete
   RUNG wire#powerrail
      { S7_Templates := "SrcType := Int" } EQ_Contact(in1 := #statStep, in2 := 40)
      wire#w1
      R_Coil( #statConfigHold[11] )
      R_Coil( #statConfigHold[12] )
      R_Coil( #statConfigHold[13] )
   END_RUNG
   RUNG wire#w1
      R_Coil( #statConfigBusy )
   END_RUNG
   RUNG wire#w1
      { S7_Templates := "time_type := Time" } #statTonTimer[40].TON(pt := T#100ms, et =>)
      Move(in := 0, out1 => #statStep)
   END_RUNG
   // the same network as SCL:
   #_w1 := #statStep = 40;
   IF #_w1 THEN
       #statConfigHold[11] := FALSE;
       #statConfigHold[12] := FALSE;
       #statConfigHold[13] := FALSE;
       #statConfigBusy := FALSE;
   END_IF;
   #statTonTimer[40].TON(IN := #_w1, PT := T#100ms);
   IF #statTonTimer[40].Q THEN #statStep := 0; END_IF;
END_REGION

REGION Network 16: Servo Auto
   RUNG wire#powerrail
      Contact( #enable )
      wire#w1
      I_Contact( #enableManualCmds )
      wire#w2
      Coil( #statMonitoring.profinetOutput.AUTO )
   END_RUNG
   RUNG wire#w1
      { S7_Templates := "SrcType := Int" } NE_Contact(in1 := #statStep, in2 := 0)
   END_RUNG wire#w2
   // the same network as SCL:
   #statMonitoring.profinetOutput.AUTO := #enable AND (NOT #enableManualCmds OR (#statStep <> 0));
END_REGION

REGION Network 17: Servo Error Reset
   RUNG wire#powerrail
      Contact( #error )
      Contact( #enable )
      wire#w1
      Contact( #enableManualCmds )
      Contact( #moduleInterface.command.errorAck )
      wire#w2
      Coil( #statMonitoring.profinetOutput."ACK-ADMIN" )
   END_RUNG
   RUNG wire#w1
      I_Contact( #enableManualCmds )
      Contact( #controlNode.command.errorAck )
   END_RUNG wire#w2
   // the same network as SCL:
   #statMonitoring.profinetOutput."ACK-ADMIN" := #error AND #enable AND ((#enableManualCmds AND #moduleInterface.command.errorAck) OR (NOT #enableManualCmds AND #controlNode.command.errorAck));
END_REGION

REGION Network 18: Servo Enable
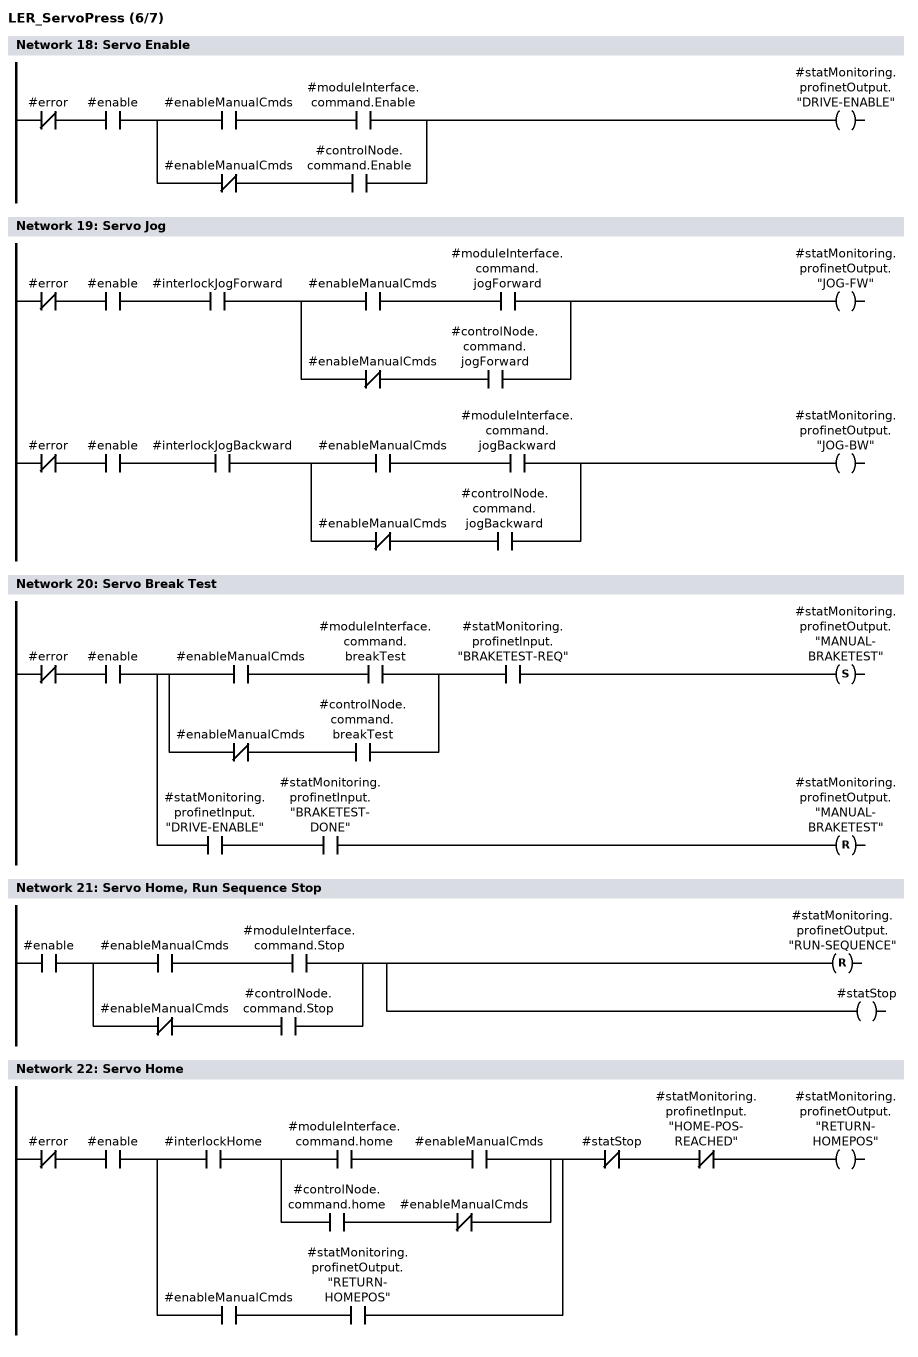
   RUNG wire#powerrail
      I_Contact( #error )
      Contact( #enable )
      wire#w1
      Contact( #enableManualCmds )
      Contact( #moduleInterface.command.Enable )
      wire#w2
      Coil( #statMonitoring.profinetOutput."DRIVE-ENABLE" )
   END_RUNG
   RUNG wire#w1
      I_Contact( #enableManualCmds )
      Contact( #controlNode.command.Enable )
   END_RUNG wire#w2
   // the same network as SCL:
   #statMonitoring.profinetOutput."DRIVE-ENABLE" := NOT #error AND #enable AND ((#enableManualCmds AND #moduleInterface.command.Enable) OR (NOT #enableManualCmds AND #controlNode.command.Enable));
END_REGION

REGION Network 19: Servo Jog
   RUNG wire#powerrail
      I_Contact( #error )
      Contact( #enable )
      Contact( #interlockJogForward )
      wire#w1
      Contact( #enableManualCmds )
      Contact( #moduleInterface.command.jogForward )
      wire#w2
      Coil( #statMonitoring.profinetOutput."JOG-FW" )
   END_RUNG
   RUNG wire#w1
      I_Contact( #enableManualCmds )
      Contact( #controlNode.command.jogForward )
   END_RUNG wire#w2
   RUNG wire#powerrail
      I_Contact( #error )
      Contact( #enable )
      Contact( #interlockJogBackward )
      wire#w3
      Contact( #enableManualCmds )
      Contact( #moduleInterface.command.jogBackward )
      wire#w4
      Coil( #statMonitoring.profinetOutput."JOG-BW" )
   END_RUNG
   RUNG wire#w3
      I_Contact( #enableManualCmds )
      Contact( #controlNode.command.jogBackward )
   END_RUNG wire#w4
   // the same network as SCL:
   #statMonitoring.profinetOutput."JOG-FW" := NOT #error AND #enable AND #interlockJogForward AND ((#enableManualCmds AND #moduleInterface.command.jogForward) OR (NOT #enableManualCmds AND #controlNode.command.jogForward));
   #statMonitoring.profinetOutput."JOG-BW" := NOT #error AND #enable AND #interlockJogBackward AND ((#enableManualCmds AND #moduleInterface.command.jogBackward) OR (NOT #enableManualCmds AND #controlNode.command.jogBackward));
END_REGION

REGION Network 20: Servo Break Test
   RUNG wire#powerrail
      I_Contact( #error )
      Contact( #enable )
      wire#w1
      Contact( #enableManualCmds )
      Contact( #moduleInterface.command.breakTest )
      wire#w2
      Contact( #statMonitoring.profinetInput."BRAKETEST-REQ" )
      S_Coil( #statMonitoring.profinetOutput."MANUAL-BRAKETEST" )
   END_RUNG
   RUNG wire#w1
      I_Contact( #enableManualCmds )
      Contact( #controlNode.command.breakTest )
   END_RUNG wire#w2
   RUNG wire#w1
      Contact( #statMonitoring.profinetInput."DRIVE-ENABLE" )
      Contact( #statMonitoring.profinetInput."BRAKETEST-DONE" )
      R_Coil( #statMonitoring.profinetOutput."MANUAL-BRAKETEST" )
   END_RUNG
   // the same network as SCL:
   #_w1 := NOT #error AND #enable;
   IF #_w1 AND ((#enableManualCmds AND #moduleInterface.command.breakTest) OR (NOT #enableManualCmds AND #controlNode.command.breakTest)) AND #statMonitoring.profinetInput."BRAKETEST-REQ" THEN
       #statMonitoring.profinetOutput."MANUAL-BRAKETEST" := TRUE;
   END_IF;
   IF #_w1 AND #statMonitoring.profinetInput."DRIVE-ENABLE" AND #statMonitoring.profinetInput."BRAKETEST-DONE" THEN
       #statMonitoring.profinetOutput."MANUAL-BRAKETEST" := FALSE;
   END_IF;
END_REGION

REGION Network 21: Servo Home, Run Sequence Stop
   RUNG wire#powerrail
      Contact( #enable )
      wire#w1
      Contact( #enableManualCmds )
      Contact( #moduleInterface.command.Stop )
      wire#w2
      R_Coil( #statMonitoring.profinetOutput."RUN-SEQUENCE" )
   END_RUNG
   RUNG wire#w1
      I_Contact( #enableManualCmds )
      Contact( #controlNode.command.Stop )
   END_RUNG wire#w2
   RUNG wire#w2
      Coil( #statStop )
   END_RUNG
   // the same network as SCL:
   #_w1 := #enable AND ((#enableManualCmds AND #moduleInterface.command.Stop) OR (NOT #enableManualCmds AND #controlNode.command.Stop));
   IF #_w1 THEN #statMonitoring.profinetOutput."RUN-SEQUENCE" := FALSE; END_IF;
   #statStop := #_w1;
END_REGION

REGION Network 22: Servo Home
   RUNG wire#powerrail
      I_Contact( #error )
      Contact( #enable )
      wire#w1
      Contact( #interlockHome )
      wire#w2
      Contact( #moduleInterface.command.home )
      Contact( #enableManualCmds )
      wire#w3
      I_Contact( #statStop )
      I_Contact( #statMonitoring.profinetInput."HOME-POS-REACHED" )
      Coil( #statMonitoring.profinetOutput."RETURN-HOMEPOS" )
   END_RUNG
   RUNG wire#w2
      Contact( #controlNode.command.home )
      I_Contact( #enableManualCmds )
   END_RUNG wire#w3
   RUNG wire#w1
      Contact( #enableManualCmds )
      Contact( #statMonitoring.profinetOutput."RETURN-HOMEPOS" )
   END_RUNG wire#w3
   // the same network as SCL:
   #statMonitoring.profinetOutput."RETURN-HOMEPOS" := NOT #error AND #enable AND ((#interlockHome AND ((#moduleInterface.command.home AND #enableManualCmds) OR (#controlNode.command.home AND NOT #enableManualCmds))) OR (#enableManualCmds AND #statMonitoring.profinetOutput."RETURN-HOMEPOS")) AND NOT #statStop AND NOT #statMonitoring.profinetInput."HOME-POS-REACHED";
END_REGION

REGION Network 23: Servo Run Sequence Start
   // #statMonitoring.profinetInput."SEQUENCE-END"
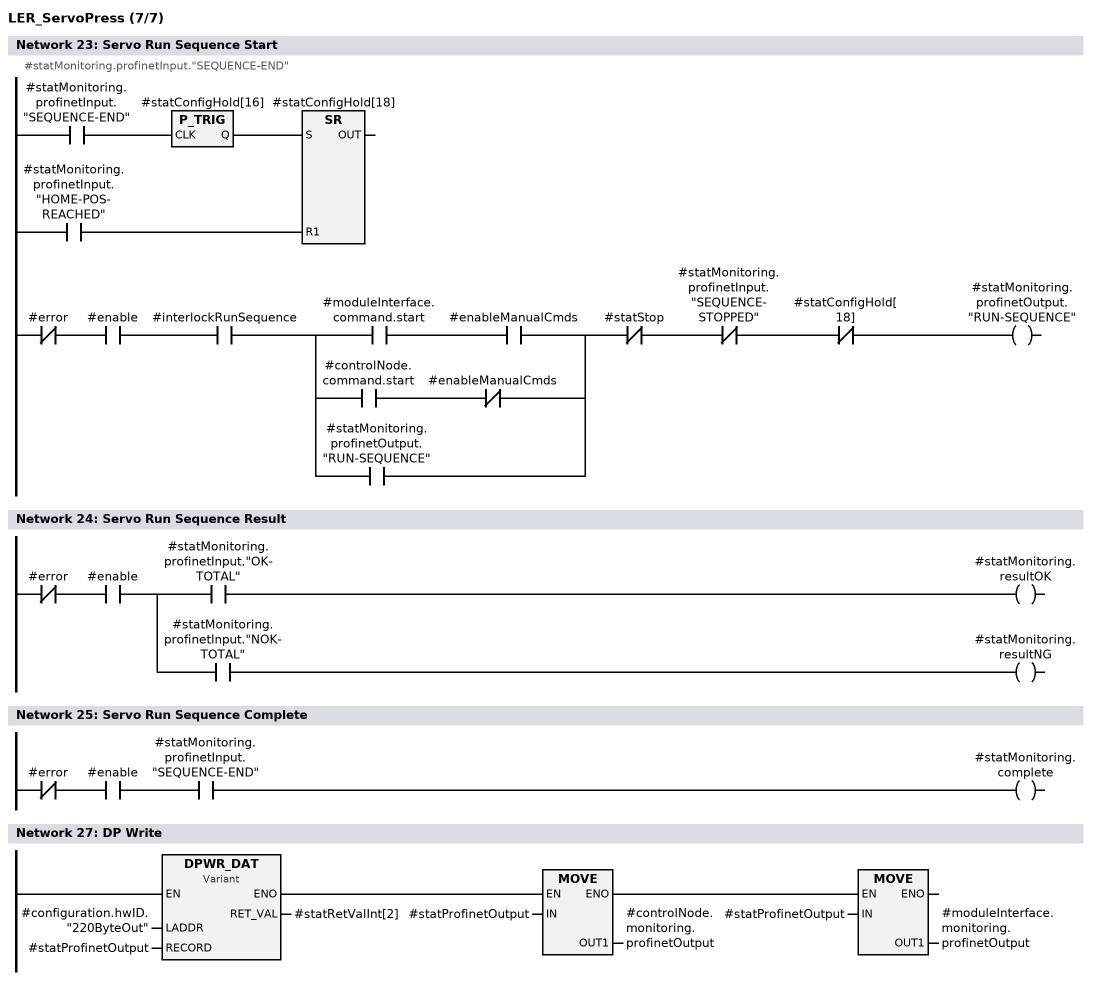
   RUNG wire#powerrail
      Contact( #statMonitoring.profinetInput."SEQUENCE-END" )
      P_Trig( #statConfigHold[16] )
      S_SR(operand := #statConfigHold[18], r1 := wire#w1)
   END_RUNG
   RUNG wire#powerrail
      Contact( #statMonitoring.profinetInput."HOME-POS-REACHED" )
   END_RUNG wire#w1
   RUNG wire#powerrail
      I_Contact( #error )
      Contact( #enable )
      Contact( #interlockRunSequence )
      wire#w2
      Contact( #moduleInterface.command.start )
      Contact( #enableManualCmds )
      wire#w3
      I_Contact( #statStop )
      I_Contact( #statMonitoring.profinetInput."SEQUENCE-STOPPED" )
      I_Contact( #statConfigHold[18] )
      Coil( #statMonitoring.profinetOutput."RUN-SEQUENCE" )
   END_RUNG
   RUNG wire#w2
      Contact( #controlNode.command.start )
      I_Contact( #enableManualCmds )
   END_RUNG wire#w3
   RUNG wire#w2
      Contact( #statMonitoring.profinetOutput."RUN-SEQUENCE" )
   END_RUNG wire#w3
   // the same network as SCL:
   #_w1 := #statMonitoring.profinetInput."SEQUENCE-END" AND NOT #statConfigHold[16];   // rising edge
   #statConfigHold[16] := #statMonitoring.profinetInput."SEQUENCE-END";
   IF #_w1 THEN
       #statConfigHold[18] := TRUE;   // SR flip-flop
   END_IF;
   IF #statMonitoring.profinetInput."HOME-POS-REACHED" THEN #statConfigHold[18] := FALSE; END_IF;
   #statMonitoring.profinetOutput."RUN-SEQUENCE" := NOT #error AND #enable AND #interlockRunSequence AND ((#moduleInterface.command.start AND #enableManualCmds) OR (#controlNode.command.start AND NOT #enableManualCmds) OR #statMonitoring.profinetOutput."RUN-SEQUENCE") AND NOT #statStop AND NOT #statMonitoring.profinetInput."SEQUENCE-STOPPED" AND NOT #statConfigHold[18];
END_REGION

REGION Network 24: Servo Run Sequence Result
   RUNG wire#powerrail
      I_Contact( #error )
      Contact( #enable )
      wire#w1
      Contact( #statMonitoring.profinetInput."OK-TOTAL" )
      Coil( #statMonitoring.resultOK )
   END_RUNG
   RUNG wire#w1
      Contact( #statMonitoring.profinetInput."NOK-TOTAL" )
      Coil( #statMonitoring.resultNG )
   END_RUNG
   // the same network as SCL:
   #_w1 := NOT #error AND #enable;
   #statMonitoring.resultOK := #_w1 AND #statMonitoring.profinetInput."OK-TOTAL";
   #statMonitoring.resultNG := #_w1 AND #statMonitoring.profinetInput."NOK-TOTAL";
END_REGION

REGION Network 25: Servo Run Sequence Complete
   RUNG wire#powerrail
      I_Contact( #error )
      Contact( #enable )
      Contact( #statMonitoring.profinetInput."SEQUENCE-END" )
      Coil( #statMonitoring.complete )
   END_RUNG
   // the same network as SCL:
   #statMonitoring.complete := NOT #error AND #enable AND #statMonitoring.profinetInput."SEQUENCE-END";
END_REGION

REGION Network 26 (SCL): Output mapping
   REGION Output mapping

       #statMonitoring.Position := #statMonitoring.profinetInput.measValueX;
       #statMonitoring.Torque := #statMonitoring.profinetInput.measValueY;
       #statMonitoring.ErrorCode :=#status;
       #statMonitoring.Start := #statMonitoring.profinetInput.START;
       #statMonitoring.Stop := #statMonitoring.profinetInput.STANDSTILL;
       #statMonitoring.Enable := #statMonitoring.profinetInput."DRIVE-ENABLE";
       #statMonitoring.busy := #statMonitoring.profinetInput."RUN-SEQUENCE" OR #statMonitoring.profinetInput."JOG-FW" OR #statMonitoring.profinetInput."JOG-BW";
       #statMonitoring.Forward := #statMonitoring.profinetInput."JOG-FW";
       #statMonitoring.Backward := #statMonitoring.profinetInput."JOG-BW";
       #statMonitoring.error := #error;

       #controlNode.monitoring.paraPV := #moduleInterface.monitoring.paraPV := #statMonitoring.paraPV;
       #controlNode.monitoring.Position := #moduleInterface.monitoring.Position := #statMonitoring.Position;
       #controlNode.monitoring.Torque := #moduleInterface.monitoring.Torque := #statMonitoring.Torque;
       #controlNode.monitoring.ErrorCode := #moduleInterface.monitoring.ErrorCode := #statMonitoring.ErrorCode;
       #controlNode.monitoring.Start := #moduleInterface.monitoring.Start := #statMonitoring.Start;
       #controlNode.monitoring.Stop := #moduleInterface.monitoring.Stop := #statMonitoring.Stop;
       #controlNode.monitoring.Enable := #moduleInterface.monitoring.Enable := #statMonitoring.Enable;
       #controlNode.monitoring.busy := #moduleInterface.monitoring.busy := #statMonitoring.busy;
       #controlNode.monitoring.complete := #moduleInterface.monitoring.complete := #statMonitoring.complete;
       #controlNode.monitoring.resultOK := #moduleInterface.monitoring.resultOK := #statMonitoring.resultOK;
       #controlNode.monitoring.resultNG := #moduleInterface.monitoring.resultNG := #statMonitoring.resultNG;
       #controlNode.monitoring.refHomeDone := #moduleInterface.monitoring.refHomeDone := #statMonitoring.refHomeDone;
       #controlNode.monitoring.Forward := #moduleInterface.monitoring.Forward := #statMonitoring.Forward;
       #controlNode.monitoring.Backward := #moduleInterface.monitoring.Backward := #statMonitoring.Backward;
       #controlNode.monitoring.error := #moduleInterface.monitoring.error := #statMonitoring.error;

       #statProfinetOutput := #statMonitoring.profinetOutput;

   END_REGION
END_REGION

REGION Network 27: DP Write
   RUNG wire#powerrail
      { S7_Templates := "[ptr_type := Variant, laddr_type := HW_IO]" } DPWR_DAT(LADDR := #configuration.hwID."220ByteOut", RECORD := #statProfinetOutput, RET_VAL => #statRetValInt[2])
      Move(in := #statProfinetOutput, out1 => #controlNode.monitoring.profinetOutput)
      Move(in := #statProfinetOutput, out1 => #moduleInterface.monitoring.profinetOutput)
   END_RUNG
   // the same network as SCL:
   #statRetValInt[2] := DPWR_DAT(LADDR := #configuration.hwID."220ByteOut",
                           RECORD := #statProfinetOutput,
                           ENO => #_w1);
   IF #_w1 THEN
       #controlNode.monitoring.profinetOutput := #statProfinetOutput;
       #moduleInterface.monitoring.profinetOutput := #statProfinetOutput;
   END_IF;
END_REGION

REGION Network 28: ******************** UNUSED ********************
END_REGION

REGION Network 29 (SCL): Servo Alarm Status
       IF #enable THEN
           IF #statMonitoring.profinetInput.alarmState <> 0 OR
               #statMonitoring.profinetInput.alarmState_1 <> 0 OR #statMonitoring.profinetInput.alarmState_2 <> 0 OR
               #statMonitoring.profinetInput.alarmState_3 <> 0 OR #statMonitoring.profinetInput.alarmState_4 <> 0 OR
               #statMonitoring.profinetInput.alarmState_5 <> 0 THEN

               #statServoAlarm.alarmState_0[0] := #statMonitoring.profinetInput.alarmState.%X0;
               #statServoAlarm.alarmState_0[1] := #statMonitoring.profinetInput.alarmState.%X1;
               #statServoAlarm.alarmState_0[2] := #statMonitoring.profinetInput.alarmState.%X2;
               #statServoAlarm.alarmState_0[3] := #statMonitoring.profinetInput.alarmState.%X3;
               #statServoAlarm.alarmState_0[4] := #statMonitoring.profinetInput.alarmState.%X4;
               #statServoAlarm.alarmState_0[5] := #statMonitoring.profinetInput.alarmState.%X5;
               #statServoAlarm.alarmState_0[6] := #statMonitoring.profinetInput.alarmState.%X6;
               #statServoAlarm.alarmState_0[7] := #statMonitoring.profinetInput.alarmState.%X7;

               #statServoAlarm.alarmState_1[0] := #statMonitoring.profinetInput.alarmState_1.%X0;
               #statServoAlarm.alarmState_1[1] := #statMonitoring.profinetInput.alarmState_1.%X1;
               #statServoAlarm.alarmState_1[2] := #statMonitoring.profinetInput.alarmState_1.%X2;
               #statServoAlarm.alarmState_1[3] := #statMonitoring.profinetInput.alarmState_1.%X3;
               #statServoAlarm.alarmState_1[4] := #statMonitoring.profinetInput.alarmState_1.%X4;
               #statServoAlarm.alarmState_1[5] := #statMonitoring.profinetInput.alarmState_1.%X5;
               #statServoAlarm.alarmState_1[6] := #statMonitoring.profinetInput.alarmState_1.%X6;
               #statServoAlarm.alarmState_1[7] := #statMonitoring.profinetInput.alarmState_1.%X7;

               #statServoAlarm.alarmState_2[0] := #statMonitoring.profinetInput.alarmState_2.%X0;
               #statServoAlarm.alarmState_2[1] := #statMonitoring.profinetInput.alarmState_2.%X1;
               #statServoAlarm.alarmState_2[2] := #statMonitoring.profinetInput.alarmState_2.%X2;
               #statServoAlarm.alarmState_2[3] := #statMonitoring.profinetInput.alarmState_2.%X3;
               #statServoAlarm.alarmState_2[4] := #statMonitoring.profinetInput.alarmState_2.%X4;
               #statServoAlarm.alarmState_2[5] := #statMonitoring.profinetInput.alarmState_2.%X5;
               #statServoAlarm.alarmState_2[6] := #statMonitoring.profinetInput.alarmState_2.%X6;
               #statServoAlarm.alarmState_2[7] := #statMonitoring.profinetInput.alarmState_2.%X7;

               #statServoAlarm.alarmState_3[0] := #statMonitoring.profinetInput.alarmState_3.%X0;
               #statServoAlarm.alarmState_3[1] := #statMonitoring.profinetInput.alarmState_3.%X1;
               #statServoAlarm.alarmState_3[2] := #statMonitoring.profinetInput.alarmState_3.%X2;
               #statServoAlarm.alarmState_3[3] := #statMonitoring.profinetInput.alarmState_3.%X3;
               #statServoAlarm.alarmState_3[4] := #statMonitoring.profinetInput.alarmState_3.%X4;
               #statServoAlarm.alarmState_3[5] := #statMonitoring.profinetInput.alarmState_3.%X5;
               #statServoAlarm.alarmState_3[6] := #statMonitoring.profinetInput.alarmState_3.%X6;
               #statServoAlarm.alarmState_3[7] := #statMonitoring.profinetInput.alarmState_3.%X7;

               #statServoAlarm.alarmState_4[0] := #statMonitoring.profinetInput.alarmState_4.%X0;
               #statServoAlarm.alarmState_4[1] := #statMonitoring.profinetInput.alarmState_4.%X1;
               #statServoAlarm.alarmState_4[2] := #statMonitoring.profinetInput.alarmState_4.%X2;
               #statServoAlarm.alarmState_4[3] := #statMonitoring.profinetInput.alarmState_4.%X3;
               #statServoAlarm.alarmState_4[4] := #statMonitoring.profinetInput.alarmState_4.%X4;
               #statServoAlarm.alarmState_4[5] := #statMonitoring.profinetInput.alarmState_4.%X5;
               #statServoAlarm.alarmState_4[6] := #statMonitoring.profinetInput.alarmState_4.%X6;
               #statServoAlarm.alarmState_4[7] := #statMonitoring.profinetInput.alarmState_4.%X7;

               #statServoAlarm.alarmState_5[0] := #statMonitoring.profinetInput.alarmState_5.%X0;
               #statServoAlarm.alarmState_5[1] := #statMonitoring.profinetInput.alarmState_5.%X1;
               #statServoAlarm.alarmState_5[2] := #statMonitoring.profinetInput.alarmState_5.%X2;
               #statServoAlarm.alarmState_5[3] := #statMonitoring.profinetInput.alarmState_5.%X3;
               #statServoAlarm.alarmState_5[4] := #statMonitoring.profinetInput.alarmState_5.%X4;
               #statServoAlarm.alarmState_5[5] := #statMonitoring.profinetInput.alarmState_5.%X5;
               #statServoAlarm.alarmState_5[6] := #statMonitoring.profinetInput.alarmState_5.%X6;
               #statServoAlarm.alarmState_5[7] := #statMonitoring.profinetInput.alarmState_5.%X7;
           END_IF;
       END_IF;
END_REGION
END_FUNCTION_BLOCK
